Staubli VAL3: BoolMess_Edit.pgx

public program BoolMess_Edit(bool& x_bRes, num x_nX, num x_nY, num x_nLength, string& x_sMess[])
  local num l_nNum
begin


   l_nNum=sel(x_bRes,1,0)
   call Sel_Edit(l_nNum,x_nX,x_nY,x_sMess)
   x_bRes=(l_nNum==1)

end
